// TIA Portal project "ArranqueTurbina" (V17)

(* hardware
DEVICE "S7-1500/ET200MP station_1"  S7-1500 station
   slot 0: "Rail_0"  Rack  6ES7 590-1***0-0AA0
   slot 1: "PLC_1"  CPU 1511-1 PN  6ES7 511-1AK02-0AB0  V2.9
      slot 3: "CPU display_1"  6ES7591-1AA00-0AA0
      slot 32768: "PROFINET interface_1"  X1
         slot 32769: "Port_1"  X1 P1
         slot 32770: "Port_2"  X1 P2
      slot 34817: "Virtual CP interface port_1"  Virtual CP interface port  Virtual CP interface port
   slot 2: "DI 16x24VDC BA_1"  DI 16x24VDC BA  6ES7 521-1BH10-0AA0  V1.1
   slot 3: "DQ 16x230VAC/2A ST_1"  DQ 16x230VAC/2A ST  6ES7 522-5HH00-0AB0  V1.1
   slot 4: "AI 4xU/I/RTD/TC ST_1"  AI 4xU/I/RTD/TC ST  6ES7 531-7QD00-0AB0  V1.0
   slot 5: "AQ 4xU/I ST_1"  AQ 4xU/I ST  6ES7 532-5HD00-0AB0  V2.2
*)

// ===== PLC "PLC_1"  CPU 1511-1 PN =====

VAR_GLOBAL   // PLC tag table "Default tag table"
   "System_Byte" AT %MB1 : Byte;
   "FirstScan" AT %M1.0 : Bool;
   "DiagStatusUpdate" AT %M1.1 : Bool;
   "AlwaysTRUE" AT %M1.2 : Bool;
   "AlwaysFALSE" AT %M1.3 : Bool;
   "Clock_Byte" AT %MB0 : Byte;
   "Clock_10Hz" AT %M0.0 : Bool;
   "Clock_5Hz" AT %M0.1 : Bool;
   "Clock_2.5Hz" AT %M0.2 : Bool;
   "Clock_2Hz" AT %M0.3 : Bool;
   "Clock_1.25Hz" AT %M0.4 : Bool;
   "Clock_1Hz" AT %M0.5 : Bool;
   "Clock_0.625Hz" AT %M0.6 : Bool;
   "Clock_0.5Hz" AT %M0.7 : Bool;
END_VAR

VAR_GLOBAL   // PLC tag table "DI"
   "Emergencia_L" AT %I0.0 : Bool;   // Parada de emergencia desde tablero local
   "Emergencia_R" AT %I0.1 : Bool;   // Parada de emergencia desde tablero remoto
   "Selectora_LR" AT %I0.2 : Bool;   // 0 = LOCAL ; 1 = REMOTO
   "Arranque_L" AT %I0.3 : Bool;   // Botón de arranque tablero local
   "Parada_L" AT %I0.4 : Bool;   // Botón parada controlada tablero local
   "Sensor_Q1" AT %I0.5 : Bool;   // Sensor de llama 1
   "Sensor_Q2" AT %I0.6 : Bool;   // Sensor de llama 2
   "Válvula_Prin" AT %I0.7 : Bool;   // 1 = Válvula principal de gas ABIERTA
   "Frenos_Aplicados" AT %I1.0 : Bool;   // 1 = Pastillas de freno aplicadas
END_VAR

VAR_GLOBAL   // PLC tag table "DQ"
   "CMD_Motor" AT %Q10.0 : Bool;   // Comando de arranque motor auxiliar
   "CMD_Junta" AT %Q10.1 : Bool;   // Comando acople junta neumática
   "CMD_Chispero1" AT %Q10.2 : Bool;   // Comando chispero 1
   "CMD_Chispero2" AT %Q10.3 : Bool;   // Comando chispero 2
   "CMD_Frenos" AT %Q10.4 : Bool;   // Comando frenos
   "CMD_Escape" AT %Q10.5 : Bool;   // Comando válvula de escape
   "CMD_Emergencia" AT %Q10.6 : Bool;   // Comando válvula de emergencia
   "CMD_ManualAutomático" AT %Q10.7 : Bool;   // Comando al sistema de control 0 = MANUAL ; 1 = AUTO
END_VAR

VAR_GLOBAL   // PLC tag table "AI"
   "Sensor_Velocidad" AT %IW20 : Int;   // Sensor de velocidad, 0..6000 RPM
   "Sensor_Temperatura" AT %IW22 : Int;   // Sensor de temperatura, 0..400C°
   "Sensor_Presión" AT %IW24 : Int;   // Sensor de presion, 0..6bar
END_VAR

VAR_GLOBAL   // PLC tag table "AQ"
   "SP_Velocidad" AT %QW30 : Int;   // Consigna de velocidad a controlador externo
   "SP_Manual" AT %QW32 : Int;   // Cosigna apertura manual a controlador externo
END_VAR

DATA_BLOCK "DB_Sistema"   // DB1
{ S7_Optimized_Access := 'TRUE' }
VERSION : 0.1
   VAR
      HMI : Struct
         CMD_Arranque : Bool;   // Comando de arranque desde HMI
         CMD_Parada : Bool;   // Comando de parada controlado desde HMI
      END_STRUCT;
      Lecturas : Struct
         Velocidad : Real;
         Temperatura : Real;
         Presión : Real;
      END_STRUCT;
      Paso : Array[1..6] of Bool;
      Consigna : Struct
         SP_Man_Valv : Real;
         SP_Auto_Vel : Real;
      END_STRUCT;
      Seguridad : Struct
         Parada_Controlada : Bool;
         Parada_Emergencia : Bool;
      END_STRUCT;
   END_VAR
BEGIN
END_DATA_BLOCK

DATA_BLOCK "Turbina_DB"   // DB7
{ S7_Optimized_Access := 'TRUE' }
VERSION : 0.1
// stored: InstanceOfName Turbina
"Turbina"
BEGIN
END_DATA_BLOCK

// folder: System blocks/Program resources

DATA_BLOCK "Delay_acople"   // DB2
{ S7_Optimized_Access := 'TRUE' }
AUTHOR : Simatic
FAMILY : IEC
NAME : IEC_TMR
VERSION : 1.0
// stored: InstanceOfName IEC_TIMER
"IEC_TIMER"
BEGIN
END_DATA_BLOCK

DATA_BLOCK "Delay_Chisperos"   // DB3
{ S7_Optimized_Access := 'TRUE' }
AUTHOR : Simatic
FAMILY : IEC
NAME : IEC_TMR
VERSION : 1.0
// stored: InstanceOfName IEC_TIMER
"IEC_TIMER"
BEGIN
END_DATA_BLOCK

DATA_BLOCK "Delay_Desacople"   // DB4
{ S7_Optimized_Access := 'TRUE' }
AUTHOR : Simatic
FAMILY : IEC
NAME : IEC_TMR
VERSION : 1.0
// stored: InstanceOfName IEC_TIMER
"IEC_TIMER"
BEGIN
END_DATA_BLOCK

DATA_BLOCK "Delay_ParadaCtrl"   // DB5
{ S7_Optimized_Access := 'TRUE' }
AUTHOR : Simatic
FAMILY : IEC
NAME : IEC_TMR
VERSION : 1.0
// stored: InstanceOfName IEC_TIMER
"IEC_TIMER"
BEGIN
END_DATA_BLOCK

DATA_BLOCK "Falla_Presion"   // DB6
{ S7_Optimized_Access := 'TRUE' }
AUTHOR : Simatic
FAMILY : IEC
NAME : IEC_TMR
VERSION : 1.0
// stored: InstanceOfName IEC_TIMER
"IEC_TIMER"
BEGIN
END_DATA_BLOCK

// folder: (top level)

FUNCTION_BLOCK "Turbina"   // FB1, LAD
{ S7_Optimized_Access := 'TRUE' }
VERSION : 0.1
   VAR_INPUT
      MotorAuxiliar : Bool;
      JuntaNeum : Bool;
      Frenos : Bool;
      Quemador_A : Bool;   // Entrada digital - Sensor Quemador A
      Quemador_B : Bool;   // Entrada digital - Sensor Quemador B
      Reset : Bool := false;
      ModoControl : Bool := false;   // Modo de control = 0=Manual 1=Auto
      SPManual : Int;   // Consigna manual
      SPAuto : Int := 0;   // Consigna Automatica
   END_VAR
   VAR_OUTPUT
      SalidaVel : Int;
      SalidaPres : Int;
   END_VAR
   VAR_IN_OUT
      DB_Lazo : PID_Compact;
   END_VAR
   VAR
      Comando : Real;
      VelReal : Real;
      ValvReal : Real;
      ModeloPlanta : "ModeloPlanta";
      SP_ManualReal : Real;
      Valvula : Int;
      SP_AutoReal : Real;
   END_VAR
   VAR_TEMP
      KFrenos : Real;
      KMotor : Real;
      state : Int;
      error : Bool;
   END_VAR
   VAR_TEMP   // added for the SCL form of the ladder/FBD networks
      _w1 : Bool;
   END_VAR
BEGIN

REGION Network 1
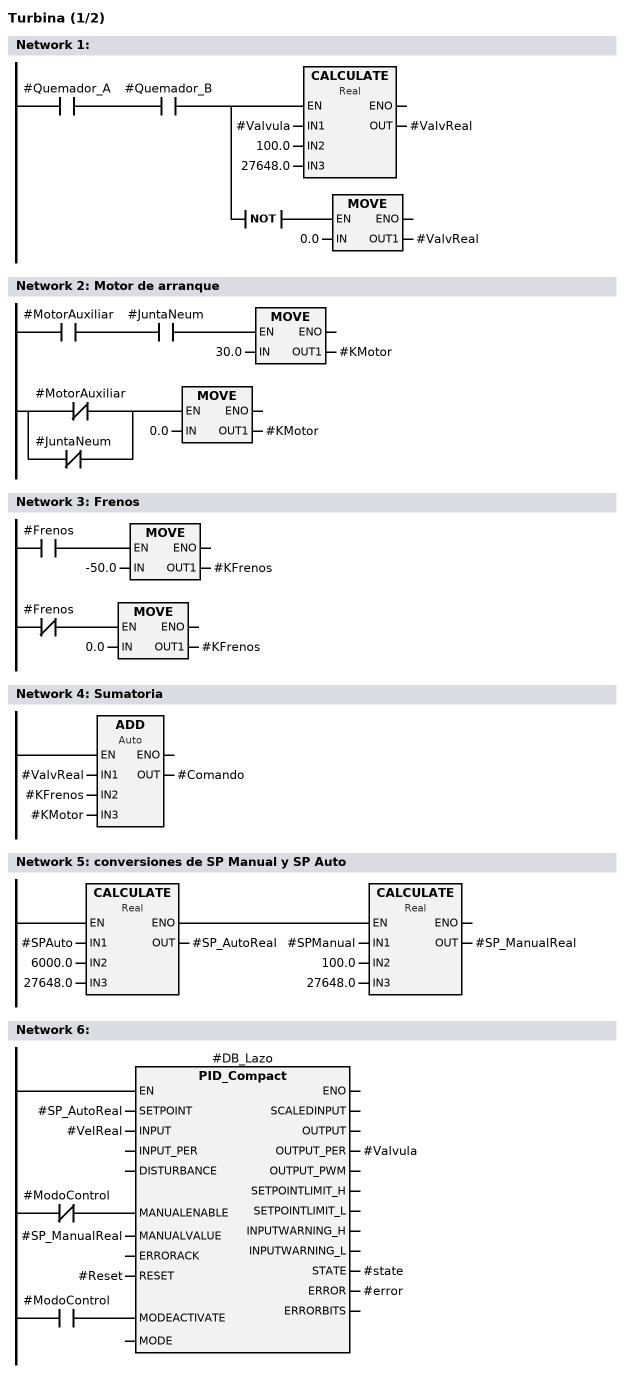
   RUNG wire#powerrail
      Contact( #Quemador_A )
      Contact( #Quemador_B )
      wire#w1
      { S7_Templates := "SrcType := Real"; S7_Expression := "(IN1*IN2)/IN3" } Calculate(in1 := #Valvula, in2 := 100.0, in3 := 27648.0, out => #ValvReal)
   END_RUNG
   RUNG wire#w1
      Not()
      Move(in := 0.0, out1 => #ValvReal)
   END_RUNG
   // the same network as SCL:
   #_w1 := #Quemador_A AND #Quemador_B;
   IF #_w1 THEN #ValvReal := (#Valvula*100.0)/27648.0; END_IF;
   IF NOT #_w1 THEN #ValvReal := 0.0; END_IF;
END_REGION

REGION Network 2: Motor de arranque
   RUNG wire#powerrail
      Contact( #MotorAuxiliar )
      Contact( #JuntaNeum )
      Move(in := 30.0, out1 => #KMotor)
   END_RUNG
   RUNG wire#powerrail
      I_Contact( #MotorAuxiliar )
      wire#w1
      Move(in := 0.0, out1 => #KMotor)
   END_RUNG
   RUNG wire#powerrail
      I_Contact( #JuntaNeum )
   END_RUNG wire#w1
   // the same network as SCL:
   IF #MotorAuxiliar AND #JuntaNeum THEN #KMotor := 30.0; END_IF;
   IF NOT #MotorAuxiliar OR NOT #JuntaNeum THEN #KMotor := 0.0; END_IF;
END_REGION

REGION Network 3: Frenos
   RUNG wire#powerrail
      Contact( #Frenos )
      Move(in := -50.0, out1 => #KFrenos)
   END_RUNG
   RUNG wire#powerrail
      I_Contact( #Frenos )
      Move(in := 0.0, out1 => #KFrenos)
   END_RUNG
   // the same network as SCL:
   IF #Frenos THEN #KFrenos := -50.0; END_IF;
   IF NOT #Frenos THEN #KFrenos := 0.0; END_IF;
END_REGION

REGION Network 4: Sumatoria
   RUNG wire#powerrail
      Add(in1 := #ValvReal, in2 := #KFrenos, in3 := #KMotor, out => #Comando)
   END_RUNG
   // the same network as SCL:
   #Comando := #ValvReal + #KFrenos + #KMotor;
END_REGION

REGION Network 5: conversiones de SP Manual y SP Auto
   RUNG wire#powerrail
      { S7_Templates := "SrcType := Real"; S7_Expression := "(IN1*IN2)/IN3" } Calculate(in1 := #SPAuto, in2 := 6000.0, in3 := 27648.0, out => #SP_AutoReal)
      { S7_Templates := "SrcType := Real"; S7_Expression := "(IN1*IN2)/IN3" } Calculate(in1 := #SPManual, in2 := 100.0, in3 := 27648.0, out => #SP_ManualReal)
   END_RUNG
   // the same network as SCL:
   #SP_AutoReal := (#SPAuto*6000.0)/27648.0;
   #SP_ManualReal := (#SPManual*100.0)/27648.0;
END_REGION

REGION Network 6
   #DB_Lazo(Setpoint := #SP_AutoReal,   // PID_Compact
            Input := #VelReal,
            ManualEnable := NOT #ModoControl,
            ManualValue := #SP_ManualReal,
            Reset := #Reset,
            ModeActivate := #ModoControl,
            Output_PER => #Valvula,
            State => #state,
            Error => #error);
END_REGION

REGION Network 7
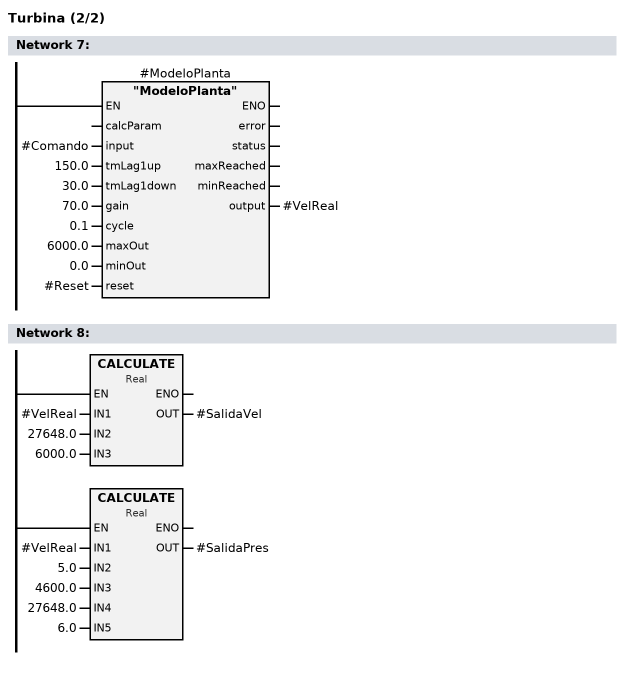
   RUNG wire#powerrail
      #ModeloPlanta(calcParam :=, input := #Comando, tmLag1up := 150.0, tmLag1down := 30.0, gain := 70.0, cycle := 0.1, maxOut := 6000.0, minOut := 0.0, reset := #Reset, error =>, status =>, maxReached =>, minReached =>, output => #VelReal)
   END_RUNG
   // the same network as SCL:
   #ModeloPlanta(input := #Comando,   // "ModeloPlanta"
                 tmLag1up := 150.0,
                 tmLag1down := 30.0,
                 gain := 70.0,
                 cycle := 0.1,
                 maxOut := 6000.0,
                 minOut := 0.0,
                 reset := #Reset,
                 output => #VelReal);
END_REGION

REGION Network 8
   RUNG wire#powerrail
      { S7_Templates := "SrcType := Real"; S7_Expression := "(IN1*IN2)/IN3" } Calculate(in1 := #VelReal, in2 := 27648.0, in3 := 6000.0, out => #SalidaVel)
   END_RUNG
   RUNG wire#powerrail
      { S7_Templates := "SrcType := Real"; S7_Expression := "(((IN1*IN2)/IN3)*IN4)/IN5" } Calculate(in1 := #VelReal, in2 := 5.0, in3 := 4600.0, in4 := 27648.0, in5 := 6.0, out => #SalidaPres)
   END_RUNG
   // the same network as SCL:
   #SalidaVel := (#VelReal*27648.0)/6000.0;
   #SalidaPres := (((#VelReal*5.0)/4600.0)*27648.0)/6.0;
END_REGION
END_FUNCTION_BLOCK

FUNCTION_BLOCK "ModeloPlanta"   // FB51, SCL
{ S7_Optimized_Access := 'TRUE' }
VERSION : 2.01
   VAR_INPUT
      calcParam : Bool;   // recalculate with new parameters
      input : Real;   // input signal
      tmLag1up : Real := 1.0;   // time constant T1 [sec] rising input
      tmLag1down : Real := 10.0;   // time constant T1 [sec] falling input
      gain : Real := 1.0;   // gain factor
      cycle : Real := 0.1;   // cyclic time [sec]
      maxOut : Real := 100.0;   // max. output limit
      minOut : Real;   // min. output limit
      reset : Bool;   // resets all relevant parameters to ‘0’ including the output
   END_VAR
   VAR_OUTPUT
      error : Bool;   // error (#tmLag1 <= 0 or #tmLag2 <= 0)
      status : Word;   // status (if #error = TRUE then status = 16#8001)
      maxReached : Bool;   // output has reached max. limit
      minReached : Bool;   // output has reached min. limit
      output : Real;   // output signal (if #error = FALSE)
   END_VAR
   VAR
      statRxn1 : Real;   // delayed input signal (n-1)
      statRyn1 : Real;   // delayed output signal (n-1)
      statRf1up : Real;   // Z-parameter 1 (rising xn)
      statRe1up : Real;   // Z-parameter 2 (rising xn)
      statRf1dn : Real;   // Z-parameter 1 (falling xn)
      statRe1dn : Real;   // Z-parameter 2 (falling xn)
      statRf1 : Real;   // active Z-parameter 1
      statRe1 : Real;   // active Z-parameter 2
      statOverfirst : Bool;
      statOutput : Real;
   END_VAR
BEGIN
   //=============================================================================
   //SIEMENS AG
   //(c)Copyright 2017 All Rights Reserved
   //-----------------------------------------------------------------------------
   //Library:       Library for Controlled System Simulation
   //Tested with:   S7-1500 FW V2.0 / S7-1200 FW V4.2
   //Engineering:   STEP 7 V14 Upd2 (TIA Portal)
   //Restrictions:  Cyclic interrupt
   //Requirements:  memory card needed for S7-1500
   //Functionality: Simulation of a PT1-System with two different Time-Constants
   //
   //  tmLag1up: Time-Constant for positive Inputsignal changes 
   //  tmLag1down: Time-Constant for negative Inputsignal changes
   //  
   //                gain
   //  Fup(p) = ----------------
   //           tmLag1up * p + 1
   //          
   //                    gain
   //  Fdown(p) = ------------------
   //             tmLag1down * p + 1
   //          
   //  Call the simulation in a cyclic interrupt with
   //  //  cyclic interrupt time at least = tmLag1/10!
   //-----------------------------------------------------------------------------
   //Change log table:
   //Version  Date       Expert in charge                Changes applied
   //02.00.00 03.02.2016 Siemens Industry Online Support Release (STEP 7 V13 SP1)
   //02.00.01 02.03.2017 Siemens Industry Online Support Release (STEP 7 V14)
   //=============================================================================

   // check parameter
   IF #tmLag1up <= 0 OR #tmLag1down <= 0 THEN
     #error := TRUE;
     #status := W#16#8001;     // Parameter Error
     #statOutput := 0;
     #output := 0;
     RETURN;
   ELSE
     #error := FALSE;
     #status := W#16#0000;     // no error
   END_IF;

   IF #calcParam = True OR NOT #statOverfirst THEN
     #statOverfirst:=1;
   // Z-parameters for Laplace PT1-System (rising signal change)
   #statRe1up := - EXP(-#cycle/#tmLag1up);
   #statRf1up := #gain*(1 + #statRe1up);
   // Z-parameters for Laplace PT1-System (falling signal change)
   #statRe1dn := - EXP(-#cycle/#tmLag1down);
   #statRf1dn := #gain*(1 + #statRe1dn);
   END_IF;

   // save delayed output signals
   #statRyn1:= #statOutput;

   // Change the parameter sets, dependent to Input Change
   IF (#input - #statRxn1) > 0 THEN
     #statRf1 := #statRf1up;
     #statRe1 := #statRe1up;
   ELSIF (#input - #statRxn1) < 0 THEN
      #statRf1 := #statRf1dn;
      #statRe1 := #statRe1dn;
   ELSE
     ;
   END_IF;

   // Differencial Equation of PT1-System
   #statOutput := #input*#statRf1 - #statRyn1*#statRe1;

   // save delayed input signals
   #statRxn1 := #input;

   // max limit of acutating variable
   IF #statOutput > #maxOut THEN
     #statOutput := #maxOut;
     #maxReached:= True;
   ELSE
     #maxReached := False;
   END_IF;

   // min limit of acutating variable
   IF #statOutput < #minOut THEN
     #statOutput := #minOut;
     #minReached := True;
   ELSE
     #minReached := False;
   END_IF;

   IF #reset THEN
     #statOutput := 0;
   END_IF;

   #output := #statOutput;
END_FUNCTION_BLOCK

FUNCTION "Secuencia" : Void   // FC1, LAD
{ S7_Optimized_Access := 'TRUE' }
VERSION : 0.1
   VAR_TEMP   // added for the SCL form of the ladder/FBD networks
      _w1 : Bool;
   END_VAR
BEGIN

REGION Network 1
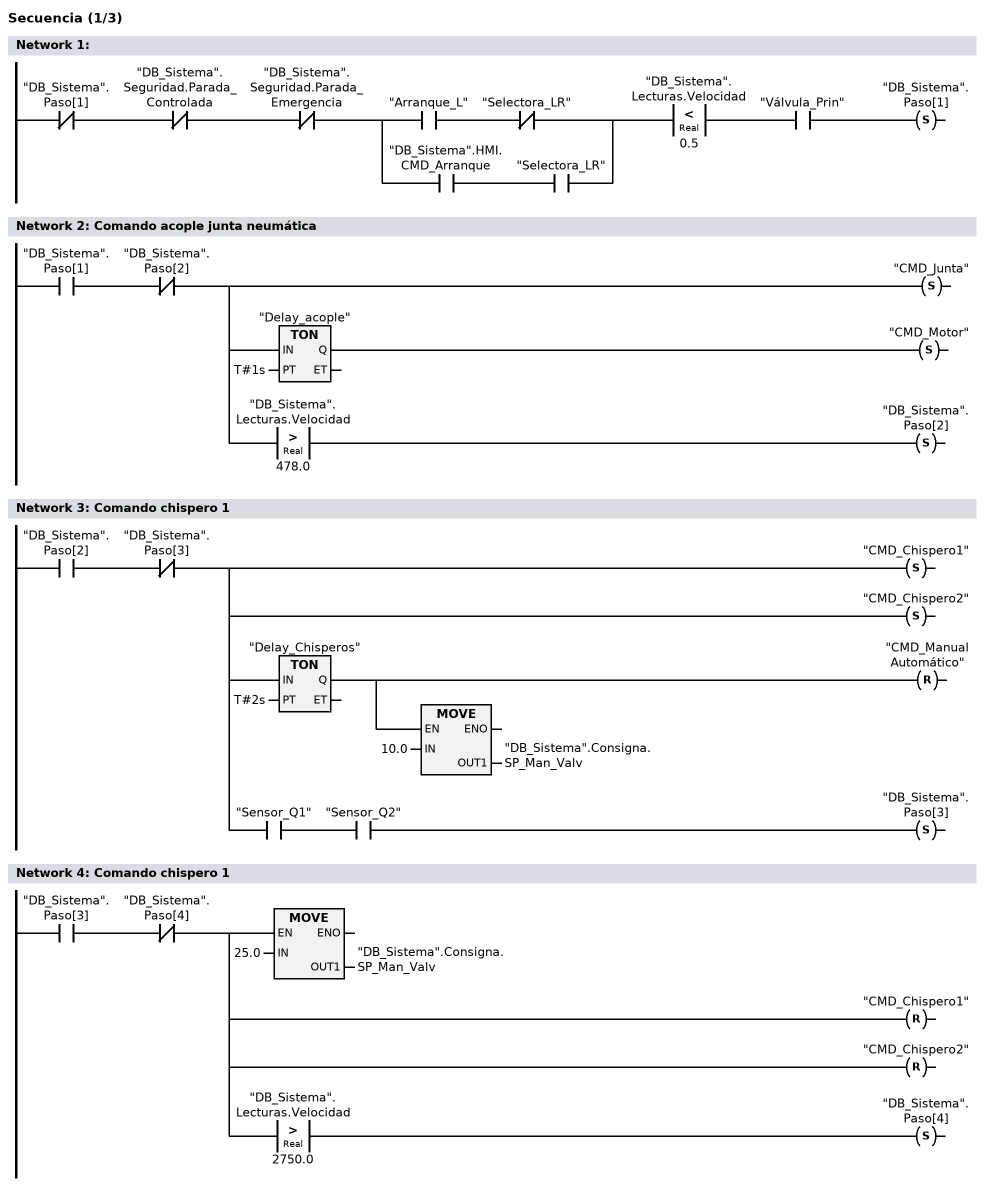
   RUNG wire#powerrail
      I_Contact( "DB_Sistema".Paso[1] )
      I_Contact( "DB_Sistema".Seguridad.Parada_Controlada )
      I_Contact( "DB_Sistema".Seguridad.Parada_Emergencia )
      wire#w1
      Contact( "Arranque_L" )
      I_Contact( "Selectora_LR" )
      wire#w2
      { S7_Templates := "SrcType := Real" } LT_Contact(in1 := "DB_Sistema".Lecturas.Velocidad, in2 := 0.5)
      Contact( "Válvula_Prin" )
      S_Coil( "DB_Sistema".Paso[1] )
   END_RUNG
   RUNG wire#w1
      Contact( "DB_Sistema".HMI.CMD_Arranque )
      Contact( "Selectora_LR" )
   END_RUNG wire#w2
   // the same network as SCL:
   IF NOT "DB_Sistema".Paso[1] AND NOT "DB_Sistema".Seguridad.Parada_Controlada AND NOT "DB_Sistema".Seguridad.Parada_Emergencia AND (("Arranque_L" AND NOT "Selectora_LR") OR ("DB_Sistema".HMI.CMD_Arranque AND "Selectora_LR")) AND ("DB_Sistema".Lecturas.Velocidad < 0.5) AND "Válvula_Prin" THEN
       "DB_Sistema".Paso[1] := TRUE;
   END_IF;
END_REGION

REGION Network 2: Comando acople junta neumática
   #_w1 := "DB_Sistema".Paso[1] AND NOT "DB_Sistema".Paso[2];
   IF #_w1 THEN "CMD_Junta" := TRUE; END_IF;
   "Delay_acople".TON(IN := #_w1, PT := T#1s);
   IF "Delay_acople".Q THEN "CMD_Motor" := TRUE; END_IF;
   IF #_w1 AND ("DB_Sistema".Lecturas.Velocidad > 478.0) THEN "DB_Sistema".Paso[2] := TRUE; END_IF;
END_REGION

REGION Network 3: Comando chispero 1
   #_w1 := "DB_Sistema".Paso[2] AND NOT "DB_Sistema".Paso[3];
   IF #_w1 THEN
       "CMD_Chispero1" := TRUE;
       "CMD_Chispero2" := TRUE;
   END_IF;
   "Delay_Chisperos".TON(IN := #_w1, PT := T#2s);
   IF "Delay_Chisperos".Q THEN
       "CMD_ManualAutomático" := FALSE;
       "DB_Sistema".Consigna.SP_Man_Valv := 10.0;
   END_IF;
   IF #_w1 AND "Sensor_Q1" AND "Sensor_Q2" THEN "DB_Sistema".Paso[3] := TRUE; END_IF;
END_REGION

REGION Network 4: Comando chispero 1
   RUNG wire#powerrail
      Contact( "DB_Sistema".Paso[3] )
      I_Contact( "DB_Sistema".Paso[4] )
      wire#w1
      Move(in := 25.0, out1 => "DB_Sistema".Consigna.SP_Man_Valv)
   END_RUNG
   RUNG wire#w1
      R_Coil( "CMD_Chispero1" )
   END_RUNG
   RUNG wire#w1
      R_Coil( "CMD_Chispero2" )
   END_RUNG
   RUNG wire#w1
      { S7_Templates := "SrcType := Real" } GT_Contact(in1 := "DB_Sistema".Lecturas.Velocidad, in2 := 2750.0)
      S_Coil( "DB_Sistema".Paso[4] )
   END_RUNG
   // the same network as SCL:
   #_w1 := "DB_Sistema".Paso[3] AND NOT "DB_Sistema".Paso[4];
   IF #_w1 THEN
       "DB_Sistema".Consigna.SP_Man_Valv := 25.0;
       "CMD_Chispero1" := FALSE;
       "CMD_Chispero2" := FALSE;
   END_IF;
   IF #_w1 AND ("DB_Sistema".Lecturas.Velocidad > 2750.0) THEN "DB_Sistema".Paso[4] := TRUE; END_IF;
END_REGION

REGION Network 5: Comando acople junta neumática
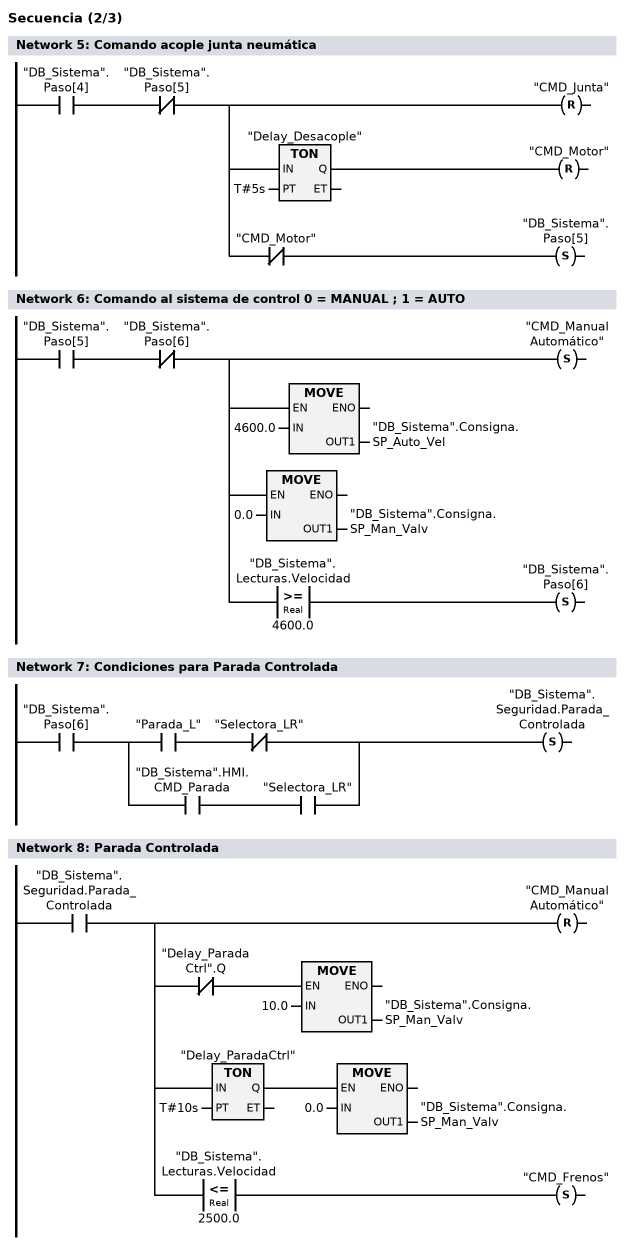
   #_w1 := "DB_Sistema".Paso[4] AND NOT "DB_Sistema".Paso[5];
   IF #_w1 THEN "CMD_Junta" := FALSE; END_IF;
   "Delay_Desacople".TON(IN := #_w1, PT := T#5s);
   IF "Delay_Desacople".Q THEN "CMD_Motor" := FALSE; END_IF;
   IF #_w1 AND NOT "CMD_Motor" THEN "DB_Sistema".Paso[5] := TRUE; END_IF;
END_REGION

REGION Network 6: Comando al sistema de control 0 = MANUAL ; 1 = AUTO
   RUNG wire#powerrail
      Contact( "DB_Sistema".Paso[5] )
      I_Contact( "DB_Sistema".Paso[6] )
      wire#w1
      S_Coil( "CMD_ManualAutomático" )
   END_RUNG
   RUNG wire#w1
      Move(in := 4600.0, out1 => "DB_Sistema".Consigna.SP_Auto_Vel)
   END_RUNG
   RUNG wire#w1
      Move(in := 0.0, out1 => "DB_Sistema".Consigna.SP_Man_Valv)
   END_RUNG
   RUNG wire#w1
      { S7_Templates := "SrcType := Real" } GE_Contact(in1 := "DB_Sistema".Lecturas.Velocidad, in2 := 4600.0)
      S_Coil( "DB_Sistema".Paso[6] )
   END_RUNG
   // the same network as SCL:
   #_w1 := "DB_Sistema".Paso[5] AND NOT "DB_Sistema".Paso[6];
   IF #_w1 THEN
       "CMD_ManualAutomático" := TRUE;
       "DB_Sistema".Consigna.SP_Auto_Vel := 4600.0;
       "DB_Sistema".Consigna.SP_Man_Valv := 0.0;
   END_IF;
   IF #_w1 AND ("DB_Sistema".Lecturas.Velocidad >= 4600.0) THEN "DB_Sistema".Paso[6] := TRUE; END_IF;
END_REGION

REGION Network 7: Condiciones para Parada Controlada
   RUNG wire#powerrail
      Contact( "DB_Sistema".Paso[6] )
      wire#w1
      Contact( "Parada_L" )
      I_Contact( "Selectora_LR" )
      wire#w2
      S_Coil( "DB_Sistema".Seguridad.Parada_Controlada )
   END_RUNG
   RUNG wire#w1
      Contact( "DB_Sistema".HMI.CMD_Parada )
      Contact( "Selectora_LR" )
   END_RUNG wire#w2
   // the same network as SCL:
   IF "DB_Sistema".Paso[6] AND (("Parada_L" AND NOT "Selectora_LR") OR ("DB_Sistema".HMI.CMD_Parada AND "Selectora_LR")) THEN
       "DB_Sistema".Seguridad.Parada_Controlada := TRUE;
   END_IF;
END_REGION

REGION Network 8: Parada Controlada
   IF "DB_Sistema".Seguridad.Parada_Controlada THEN "CMD_ManualAutomático" := FALSE; END_IF;
   IF "DB_Sistema".Seguridad.Parada_Controlada AND NOT "Delay_ParadaCtrl".Q THEN
       "DB_Sistema".Consigna.SP_Man_Valv := 10.0;
   END_IF;
   "Delay_ParadaCtrl".TON(IN := "DB_Sistema".Seguridad.Parada_Controlada, PT := T#10s);
   IF "Delay_ParadaCtrl".Q THEN "DB_Sistema".Consigna.SP_Man_Valv := 0.0; END_IF;
   IF "DB_Sistema".Seguridad.Parada_Controlada AND ("DB_Sistema".Lecturas.Velocidad <= 2500.0) THEN
       "CMD_Frenos" := TRUE;
   END_IF;
END_REGION

REGION Network 9: Reinicio Secuencia
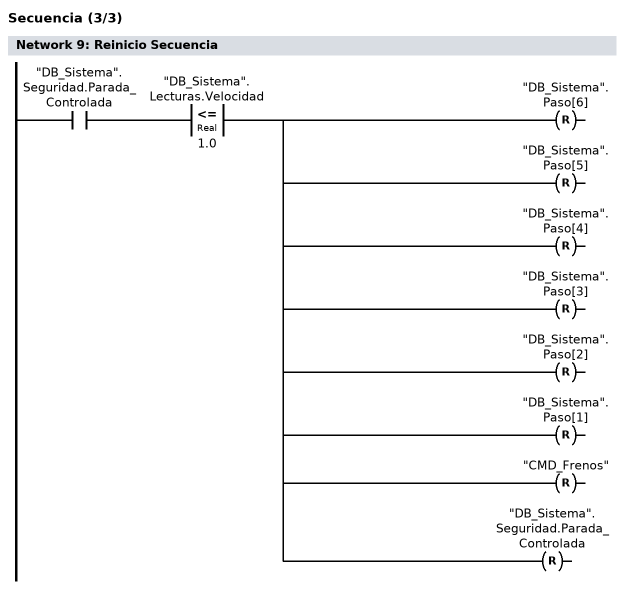
   RUNG wire#powerrail
      Contact( "DB_Sistema".Seguridad.Parada_Controlada )
      { S7_Templates := "SrcType := Real" } LE_Contact(in1 := "DB_Sistema".Lecturas.Velocidad, in2 := 1.0)
      wire#w1
      R_Coil( "DB_Sistema".Paso[6] )
   END_RUNG
   RUNG wire#w1
      R_Coil( "DB_Sistema".Paso[5] )
   END_RUNG
   RUNG wire#w1
      R_Coil( "DB_Sistema".Paso[4] )
   END_RUNG
   RUNG wire#w1
      R_Coil( "DB_Sistema".Paso[3] )
   END_RUNG
   RUNG wire#w1
      R_Coil( "DB_Sistema".Paso[2] )
   END_RUNG
   RUNG wire#w1
      R_Coil( "DB_Sistema".Paso[1] )
   END_RUNG
   RUNG wire#w1
      R_Coil( "CMD_Frenos" )
   END_RUNG
   RUNG wire#w1
      R_Coil( "DB_Sistema".Seguridad.Parada_Controlada )
   END_RUNG
   // the same network as SCL:
   IF "DB_Sistema".Seguridad.Parada_Controlada AND ("DB_Sistema".Lecturas.Velocidad <= 1.0) THEN
       "DB_Sistema".Paso[6] := FALSE;
       "DB_Sistema".Paso[5] := FALSE;
       "DB_Sistema".Paso[4] := FALSE;
       "DB_Sistema".Paso[3] := FALSE;
       "DB_Sistema".Paso[2] := FALSE;
       "DB_Sistema".Paso[1] := FALSE;
       "CMD_Frenos" := FALSE;
       "DB_Sistema".Seguridad.Parada_Controlada := FALSE;
   END_IF;
END_REGION
END_FUNCTION

FUNCTION "Seguridad" : Void   // FC2, LAD
{ S7_Optimized_Access := 'TRUE' }
VERSION : 0.1
BEGIN

REGION Network 1: Indicacion Parada de Emergencia
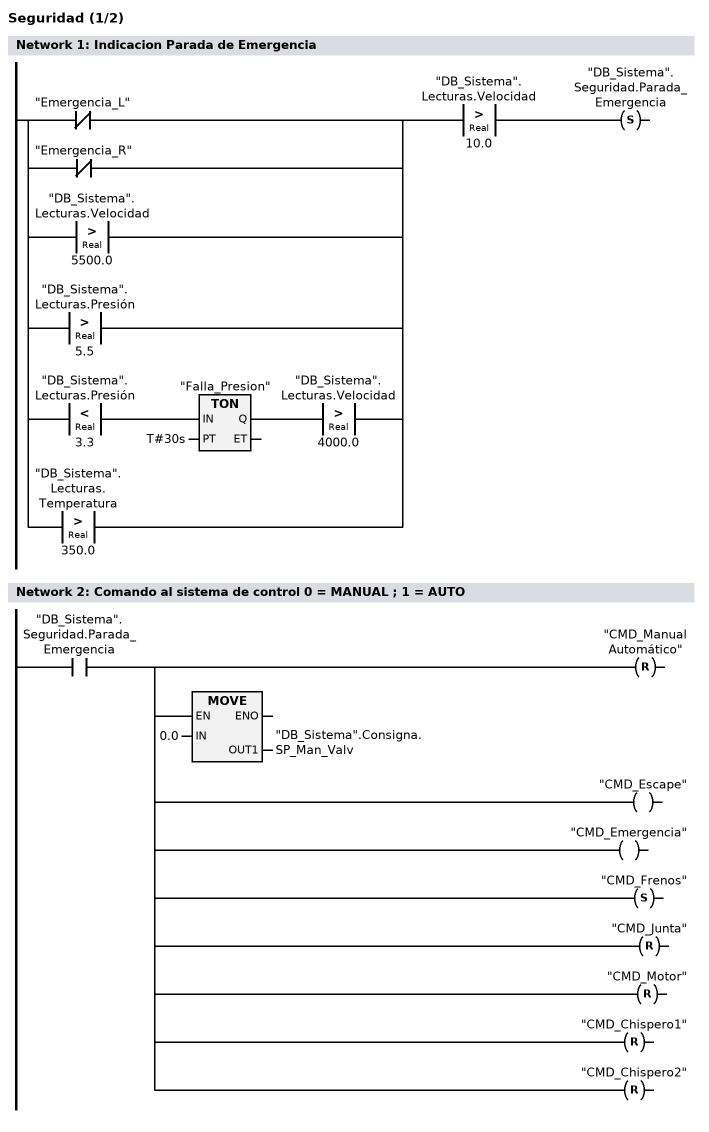
   "Falla_Presion".TON(IN := "DB_Sistema".Lecturas.Presión < 3.3, PT := T#30s);
   IF (NOT "Emergencia_L" OR NOT "Emergencia_R" OR ("DB_Sistema".Lecturas.Velocidad > 5500.0) OR ("DB_Sistema".Lecturas.Presión > 5.5) OR ("Falla_Presion".Q AND ("DB_Sistema".Lecturas.Velocidad > 4000.0)) OR ("DB_Sistema".Lecturas.Temperatura > 350.0)) AND ("DB_Sistema".Lecturas.Velocidad > 10.0) THEN
       "DB_Sistema".Seguridad.Parada_Emergencia := TRUE;
   END_IF;
END_REGION

REGION Network 2: Comando al sistema de control 0 = MANUAL ; 1 = AUTO
   RUNG wire#powerrail
      Contact( "DB_Sistema".Seguridad.Parada_Emergencia )
      wire#w1
      R_Coil( "CMD_ManualAutomático" )
   END_RUNG
   RUNG wire#w1
      Move(in := 0.0, out1 => "DB_Sistema".Consigna.SP_Man_Valv)
   END_RUNG
   RUNG wire#w1
      Coil( "CMD_Escape" )
   END_RUNG
   RUNG wire#w1
      Coil( "CMD_Emergencia" )
   END_RUNG
   RUNG wire#w1
      S_Coil( "CMD_Frenos" )
   END_RUNG
   RUNG wire#w1
      R_Coil( "CMD_Junta" )
   END_RUNG
   RUNG wire#w1
      R_Coil( "CMD_Motor" )
   END_RUNG
   RUNG wire#w1
      R_Coil( "CMD_Chispero1" )
   END_RUNG
   RUNG wire#w1
      R_Coil( "CMD_Chispero2" )
   END_RUNG
   // the same network as SCL:
   IF "DB_Sistema".Seguridad.Parada_Emergencia THEN
       "CMD_ManualAutomático" := FALSE;
       "DB_Sistema".Consigna.SP_Man_Valv := 0.0;
   END_IF;
   "CMD_Escape" := "DB_Sistema".Seguridad.Parada_Emergencia;
   "CMD_Emergencia" := "DB_Sistema".Seguridad.Parada_Emergencia;
   IF "DB_Sistema".Seguridad.Parada_Emergencia THEN
       "CMD_Frenos" := TRUE;
       "CMD_Junta" := FALSE;
       "CMD_Motor" := FALSE;
       "CMD_Chispero1" := FALSE;
       "CMD_Chispero2" := FALSE;
   END_IF;
END_REGION

REGION Network 3: Reinicio Secuencia
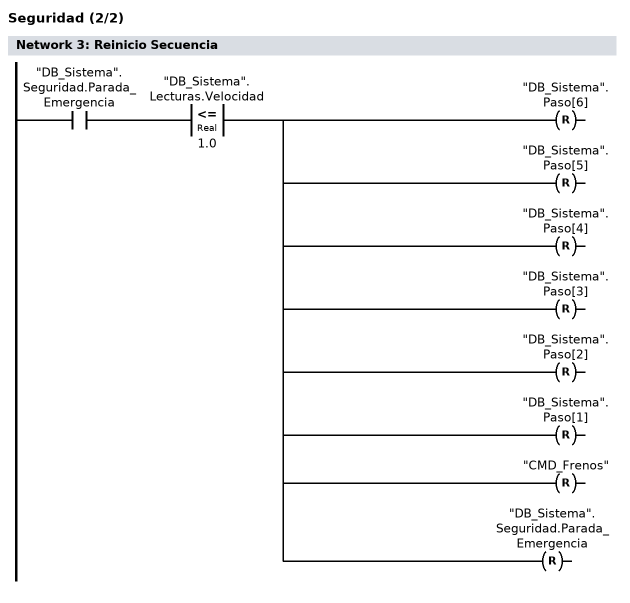
   RUNG wire#powerrail
      Contact( "DB_Sistema".Seguridad.Parada_Emergencia )
      { S7_Templates := "SrcType := Real" } LE_Contact(in1 := "DB_Sistema".Lecturas.Velocidad, in2 := 1.0)
      wire#w1
      R_Coil( "DB_Sistema".Paso[6] )
   END_RUNG
   RUNG wire#w1
      R_Coil( "DB_Sistema".Paso[5] )
   END_RUNG
   RUNG wire#w1
      R_Coil( "DB_Sistema".Paso[4] )
   END_RUNG
   RUNG wire#w1
      R_Coil( "DB_Sistema".Paso[3] )
   END_RUNG
   RUNG wire#w1
      R_Coil( "DB_Sistema".Paso[2] )
   END_RUNG
   RUNG wire#w1
      R_Coil( "DB_Sistema".Paso[1] )
   END_RUNG
   RUNG wire#w1
      R_Coil( "CMD_Frenos" )
   END_RUNG
   RUNG wire#w1
      R_Coil( "DB_Sistema".Seguridad.Parada_Emergencia )
   END_RUNG
   // the same network as SCL:
   IF "DB_Sistema".Seguridad.Parada_Emergencia AND ("DB_Sistema".Lecturas.Velocidad <= 1.0) THEN
       "DB_Sistema".Paso[6] := FALSE;
       "DB_Sistema".Paso[5] := FALSE;
       "DB_Sistema".Paso[4] := FALSE;
       "DB_Sistema".Paso[3] := FALSE;
       "DB_Sistema".Paso[2] := FALSE;
       "DB_Sistema".Paso[1] := FALSE;
       "CMD_Frenos" := FALSE;
       "DB_Sistema".Seguridad.Parada_Emergencia := FALSE;
   END_IF;
END_REGION
END_FUNCTION

FUNCTION "Escalado_AI" : Void   // FC3, LAD
{ S7_Optimized_Access := 'TRUE' }
VERSION : 0.1
   VAR_INPUT
      Sensor : Int;
      MAX_Sensor : Real;
      MIN_Sensor : Real;
      MAX_Canal : Int;
      MIN_Canal : Int;
   END_VAR
   VAR_OUTPUT
      Sensor_Escalado : Real;
   END_VAR
   VAR_TEMP
      Sensor_Normalizado : Real;
   END_VAR
BEGIN

REGION Network 1
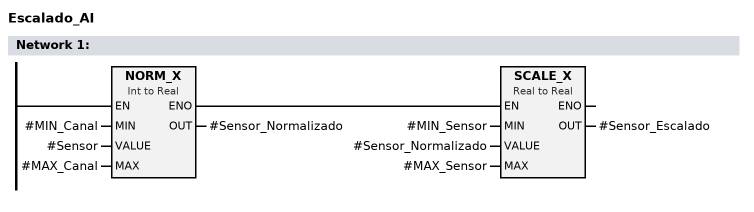
   RUNG wire#powerrail
      { S7_Templates := "[SrcType := Int, DestType := Real]" } Normalize(min := #MIN_Canal, value := #Sensor, max := #MAX_Canal, out => #Sensor_Normalizado)
      { S7_Templates := "[SrcType := Real, DestType := Real]" } Scale(min := #MIN_Sensor, value := #Sensor_Normalizado, max := #MAX_Sensor, out => #Sensor_Escalado)
   END_RUNG
   // the same network as SCL:
   #Sensor_Normalizado := NORM_X(MIN := #MIN_Canal, VALUE := #Sensor, MAX := #MAX_Canal);
   #Sensor_Escalado := SCALE_X(MIN := #MIN_Sensor, VALUE := #Sensor_Normalizado, MAX := #MAX_Sensor);
END_REGION
END_FUNCTION

FUNCTION "Escalado_AQ" : Void   // FC4, LAD
{ S7_Optimized_Access := 'TRUE' }
VERSION : 0.1
   VAR_INPUT
      Comando : Real;
      MAX_Comando : Real;
      MIN_Comando : Real;
      MAX_Actuador : Int;
      MIN_Actuador : Int;
   END_VAR
   VAR_OUTPUT
      Salida : Int;
   END_VAR
   VAR_TEMP
      Normalizado : Real;
   END_VAR
BEGIN

REGION Network 1
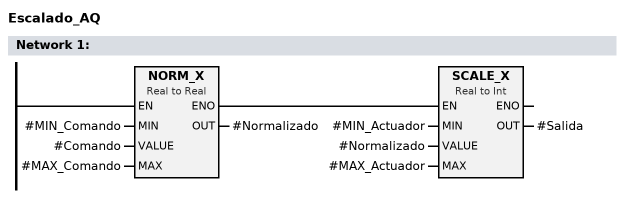
   RUNG wire#powerrail
      { S7_Templates := "[SrcType := Real, DestType := Real]" } Normalize(min := #MIN_Comando, value := #Comando, max := #MAX_Comando, out => #Normalizado)
      { S7_Templates := "[SrcType := Real, DestType := Int]" } Scale(min := #MIN_Actuador, value := #Normalizado, max := #MAX_Actuador, out => #Salida)
   END_RUNG
   // the same network as SCL:
   #Normalizado := NORM_X(MIN := #MIN_Comando, VALUE := #Comando, MAX := #MAX_Comando);
   #Salida := SCALE_X(MIN := #MIN_Actuador, VALUE := #Normalizado, MAX := #MAX_Actuador);
END_REGION
END_FUNCTION

ORGANIZATION_BLOCK "Main"   // OB1, LAD, ProgramCycle
TITLE = "Main Program Sweep (Cycle)"
{ S7_Optimized_Access := 'TRUE' }
VERSION : 0.1
   VAR_INPUT
      Initial_Call : Bool;   // Initial call of this OB
      Remanence : Bool;   // =True, if remanent data are available
   END_VAR
BEGIN

REGION Network 1
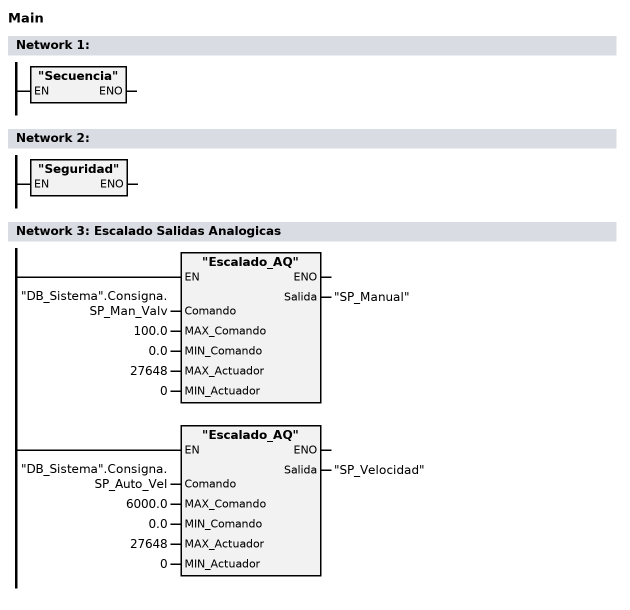
   RUNG wire#powerrail
      "Secuencia"()
   END_RUNG
   // the same network as SCL:
   "Secuencia"();
END_REGION

REGION Network 2
   RUNG wire#powerrail
      "Seguridad"()
   END_RUNG
   // the same network as SCL:
   "Seguridad"();
END_REGION

REGION Network 3: Escalado Salidas Analogicas
   RUNG wire#powerrail
      "Escalado_AQ"(Comando := "DB_Sistema".Consigna.SP_Man_Valv, MAX_Comando := 100.0, MIN_Comando := 0.0, MAX_Actuador := 27648, MIN_Actuador := 0, Salida => "SP_Manual")
   END_RUNG
   RUNG wire#powerrail
      "Escalado_AQ"(Comando := "DB_Sistema".Consigna.SP_Auto_Vel, MAX_Comando := 6000.0, MIN_Comando := 0.0, MAX_Actuador := 27648, MIN_Actuador := 0, Salida => "SP_Velocidad")
   END_RUNG
   // the same network as SCL:
   "Escalado_AQ"(Comando := "DB_Sistema".Consigna.SP_Man_Valv,
                 MAX_Comando := 100.0,
                 MIN_Comando := 0.0,
                 MAX_Actuador := 27648,
                 MIN_Actuador := 0,
                 Salida => "SP_Manual");
   "Escalado_AQ"(Comando := "DB_Sistema".Consigna.SP_Auto_Vel,
                 MAX_Comando := 6000.0,
                 MIN_Comando := 0.0,
                 MAX_Actuador := 27648,
                 MIN_Actuador := 0,
                 Salida => "SP_Velocidad");
END_REGION
END_ORGANIZATION_BLOCK

ORGANIZATION_BLOCK "Cyclic interrupt"   // OB30, LAD, CyclicInterrupt
{ S7_Optimized_Access := 'TRUE' }
VERSION : 0.1
   VAR_INPUT
      Initial_Call : Bool;   // Initial call of this OB
      Event_Count : Int;   // Events discarded
   END_VAR
BEGIN

REGION Network 1
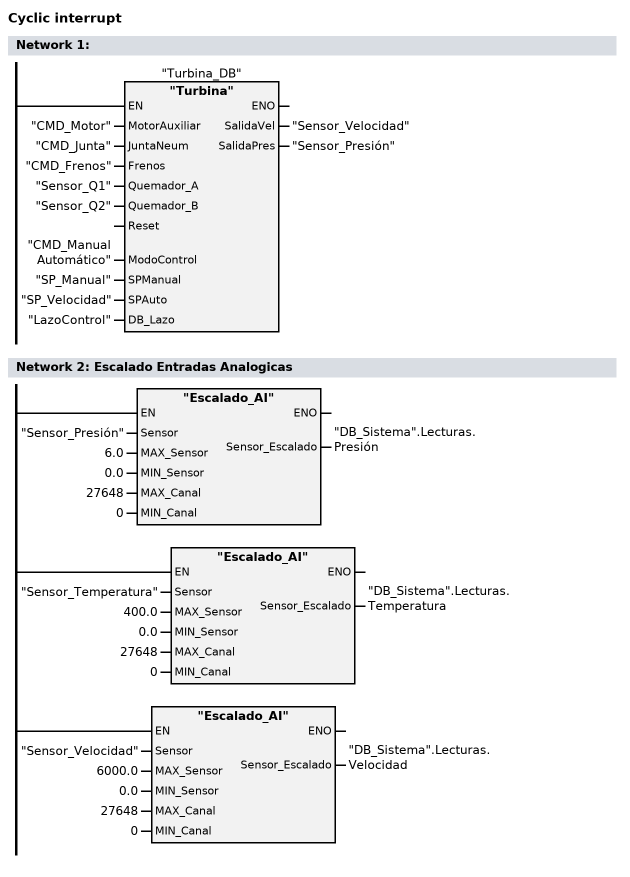
   RUNG wire#powerrail
      "Turbina_DB"(MotorAuxiliar := "CMD_Motor", JuntaNeum := "CMD_Junta", Frenos := "CMD_Frenos", Quemador_A := "Sensor_Q1", Quemador_B := "Sensor_Q2", Reset :=, ModoControl := "CMD_ManualAutomático", SPManual := "SP_Manual", SPAuto := "SP_Velocidad", DB_Lazo := "LazoControl", SalidaVel => "Sensor_Velocidad", SalidaPres => "Sensor_Presión")
   END_RUNG
   // the same network as SCL:
   "Turbina_DB"(MotorAuxiliar := "CMD_Motor",   // "Turbina"
                JuntaNeum := "CMD_Junta",
                Frenos := "CMD_Frenos",
                Quemador_A := "Sensor_Q1",
                Quemador_B := "Sensor_Q2",
                ModoControl := "CMD_ManualAutomático",
                SPManual := "SP_Manual",
                SPAuto := "SP_Velocidad",
                DB_Lazo := "LazoControl",
                SalidaVel => "Sensor_Velocidad",
                SalidaPres => "Sensor_Presión");
END_REGION

REGION Network 2: Escalado Entradas Analogicas
   RUNG wire#powerrail
      "Escalado_AI"(Sensor := "Sensor_Presión", MAX_Sensor := 6.0, MIN_Sensor := 0.0, MAX_Canal := 27648, MIN_Canal := 0, Sensor_Escalado => "DB_Sistema".Lecturas.Presión)
   END_RUNG
   RUNG wire#powerrail
      "Escalado_AI"(Sensor := "Sensor_Temperatura", MAX_Sensor := 400.0, MIN_Sensor := 0.0, MAX_Canal := 27648, MIN_Canal := 0, Sensor_Escalado => "DB_Sistema".Lecturas.Temperatura)
   END_RUNG
   RUNG wire#powerrail
      "Escalado_AI"(Sensor := "Sensor_Velocidad", MAX_Sensor := 6000.0, MIN_Sensor := 0.0, MAX_Canal := 27648, MIN_Canal := 0, Sensor_Escalado => "DB_Sistema".Lecturas.Velocidad)
   END_RUNG
   // the same network as SCL:
   "Escalado_AI"(Sensor := "Sensor_Presión",
                 MAX_Sensor := 6.0,
                 MIN_Sensor := 0.0,
                 MAX_Canal := 27648,
                 MIN_Canal := 0,
                 Sensor_Escalado => "DB_Sistema".Lecturas.Presión);
   "Escalado_AI"(Sensor := "Sensor_Temperatura",
                 MAX_Sensor := 400.0,
                 MIN_Sensor := 0.0,
                 MAX_Canal := 27648,
                 MIN_Canal := 0,
                 Sensor_Escalado => "DB_Sistema".Lecturas.Temperatura);
   "Escalado_AI"(Sensor := "Sensor_Velocidad",
                 MAX_Sensor := 6000.0,
                 MIN_Sensor := 0.0,
                 MAX_Canal := 27648,
                 MIN_Canal := 0,
                 Sensor_Escalado => "DB_Sistema".Lecturas.Velocidad);
END_REGION
END_ORGANIZATION_BLOCK